(* IEC 61131-3 sources: ml2plc/examples/models/structured_text (part 7) *)

    weights_2 : ARRAY[0..3071] OF REAL := [-0.079738, -0.018148, -0.039603, 0.086091, 0.087780, 0.006551, -0.070254, -0.061014, -0.002917, -0.104361, -0.050675, -0.028002, -0.028302, -0.113236, 0.025798, -0.042125, -0.070821, -0.030886, -0.025321, 0.020352, -0.036494, -0.007489, 0.010150, 0.002465, 0.038335, -0.010082, -0.012631, -0.130657, -0.057749, -0.014712, 0.001941, 0.017731, 0.037307, 0.060894, -0.052816, -0.038803, -0.026264, 0.004428, 0.007999, -0.071385, 0.019978, -0.025107, 0.043303, -0.056437, 0.018136, -0.004926, -0.015582, -0.040352, -0.046320, -0.051167, -0.108342, 0.061847, 0.019535, 0.024186, -0.009612, 0.051589, 0.040419, 0.004677, -0.047156, 0.011391, 0.001568, -0.006703, -0.040582, -0.044892, -0.000777, -0.114299, 0.015176, 0.022018, -0.082290, -0.099898, -0.005333, -0.000085, 0.033593, -0.100384, -0.031339, -0.014356, -0.022256, -0.006458, -0.017672, -0.016220, 0.017575, -0.003964, 0.001504, -0.101623, 0.084646, -0.162545, 0.018226, 0.046139, -0.158154, -0.011727, 0.051997, 0.013728, 0.037309, 0.037653, -0.015994, -0.013833, 0.016918, 0.072840, 0.002249, 0.021758, 0.007330, -0.005101, 0.041748, 0.049668, -0.053153, -0.059272, 0.053023, -0.004963, -0.038369, -0.042376, -0.062836, 0.007027, 0.000628, 0.064942, 0.011186, 0.136276, -0.175093, 0.033480, -0.137850, -0.093329, 0.028996, 0.027738, 0.027495, 0.066908, -0.138166, -0.062207, 0.031390, 0.016039, 0.006747, 0.041813, -0.052656, -0.001730, 0.027697, -0.081471, -0.040016, 0.029091, -0.036192, 0.076833, -0.040911, 0.054524, 0.042687, 0.004638, 0.028443, -0.015942, 0.033767, -0.010835, 0.015542, -0.054845, 0.070825, -0.016626, 0.127162, -0.148593, -0.091221, 0.026570, 0.028940, 0.004587, 0.004252, 0.003949, 0.009750, 0.054379, -0.041042, 0.045454, -0.025805, 0.023543, 0.049444, 0.016239, 0.092608, 0.023911, 0.023148, 0.032898, 0.001731, 0.000178, -0.026304, -0.012553, -0.038693, 0.011086, -0.086358, -0.012758, -0.095144, -0.067500, 0.058514, 0.063057, -0.007906, 0.011515, 0.033430, 0.059557, 0.016737, -0.005871, 0.035359, -0.028117, -0.041617, -0.050268, -0.022380, -0.027072, 0.032683, 0.043795, -0.096440, 0.061286, 0.063994, -0.063137, 0.037471, -0.013500, 0.031420, 0.048276, 0.039014, -0.015300, -0.075964, 0.020676, -0.004749, -0.019730, 0.011212, -0.001377, -0.030352, -0.032305, -0.070925, -0.009115, 0.002307, 0.015789, 0.015110, -0.050587, -0.070865, -0.040802, -0.023738, -0.059662, -0.066688, 0.087581, -0.040323, 0.046836, 0.033400, 0.041713, 0.020144, 0.004004, 0.043881, 0.012120, 0.006567, -0.047181, -0.036415, 0.020897, -0.051205, -0.018987, 0.062641, -0.077042, -0.050492, -0.009248, -0.029647, -0.028774, 0.034574, 0.026711, 0.018497, -0.078291, 0.000750, 0.036981, -0.032199, -0.046941, -0.071874, 0.018149, 0.047391, 0.036563, 0.071201, -0.046533, -0.008354, -0.010784, -0.023974, 0.000798, -0.028594, -0.005823, -0.023141, 0.052901, -0.046988, 0.042628, -0.015610, 0.017471, -0.006060, -0.071074, 0.009814, 0.028930, -0.065885, 0.004670, -0.017008, 0.040985, 0.017000, 0.023364, 0.017848, -0.010962, -0.012304, 0.056049, -0.024912, 0.058021, 0.021300, -0.043819, 0.032877, -0.103125, -0.033170, 0.024651, -0.021986, -0.040304, -0.039152, -0.070680, 0.030104, -0.009235, -0.000069, 0.079351, -0.069846, -0.013240, -0.029293, 0.010581, 0.024807, -0.148111, 0.011108, -0.006310, -0.019430, -0.007536, -0.023961, -0.058471, 0.062022, 0.030894, -0.126689, 0.014609, 0.080879, 0.077431, 0.049936, 0.057099, 0.035921, -0.095284, -0.055119, 0.003187, -0.032224, -0.023817, -0.013887, -0.012151, 0.081267, 0.002542, 0.031867, -0.038254, -0.038660, -0.020785, -0.042612, 0.006728, -0.017310, 0.096375, 0.003581, -0.078691, -0.015241, -0.028676, -0.030744, -0.033101, 0.000131, -0.012343, 0.062320, 0.038591, 0.005985, 0.042647, 0.020790, -0.148493, -0.026770, -0.021416, 0.007593, 0.007429, 0.052336, 0.045379, 0.011810, -0.062384, -0.009387, -0.031314, -0.007850, -0.031340, -0.022787, -0.021615, -0.002952, 0.056798, -0.033256, -0.040985, 0.044623, -0.019729, 0.040531, -0.009346, 0.074998, -0.115437, -0.030462, 0.063818, -0.056515, -0.067471, -0.070527, -0.068923, 0.035830, -0.052215, 0.016097, -0.058752, -0.008437, -0.024348, -0.049775, -0.009136, 0.091045, -0.007442, 0.001373, 0.006184, -0.011116, -0.078380, -0.038023, 0.059468, 0.069133, -0.014606, 0.013753, -0.061774, -0.093455, 0.029663, 0.027740, -0.001149, -0.067593, -0.015326, -0.102692, -0.049083, 0.090420, 0.002557, -0.059069, -0.012321, -0.038434, 0.014221, -0.014216, 0.018523, -0.042681, -0.041700, -0.040420, -0.076709, 0.110400, -0.077629, 0.030365, -0.005439, -0.079538, 0.055336, -0.009865, -0.003723, 0.014380, 0.023391, 0.054367, -0.023334, -0.057359, -0.021853, 0.008266, 0.039793, -0.024814, 0.010200, 0.029996, 0.015745, 0.091485, -0.035740, -0.081574, 0.032012, -0.086098, -0.021267, 0.015700, 0.026081, 0.053181, -0.011251, 0.002709, -0.017904, 0.033816, 0.041051, 0.020465, 0.044652, 0.033611, 0.034061, 0.024369, 0.022682, 0.059236, -0.037332, -0.024917, 0.081315, -0.044821, -0.039097, -0.022489, -0.018730, 0.012051, 0.015785, -0.084618, -0.059913, -0.096852, -0.002574, 0.033606, 0.032488, -0.003370, 0.021578, -0.006767, -0.090289, -0.041813, -0.130182, 0.018747, 0.026137, 0.015171, -0.023929, 0.052123, 0.021562, 0.021162, 0.021938, 0.011171, 0.021531, -0.086418, -0.003059, -0.011323, -0.022397, -0.067489, 0.024647, -0.066202, -0.063597, 0.062780, -0.004904, -0.087994, 0.028886, 0.005226, 0.009394, 0.023893, -0.172482, 0.027981, -0.000874, -0.021041, 0.003634, -0.079888, 0.033055, 0.054404, -0.056195, 0.015224, -0.133033, 0.047975, 0.015738, -0.021576, -0.054744, 0.002027, -0.013741, 0.044122, 0.026994, 0.024536, -0.007580, -0.015404, -0.107729, -0.034309, -0.001584, 0.042350, 0.027646, -0.121416, -0.070898, -0.072544, -0.011634, 0.046801, 0.015250, 0.011697, -0.042356, 0.051572, -0.065324, -0.191804, -0.028124, -0.033760, -0.010601, 0.017532, 0.028585, 0.076237, 0.019598, -0.024975, 0.031572, 0.007237, 0.067220, -0.013791, 0.011680, -0.021350, -0.002438, -0.010119, 0.007116, 0.012485, 0.033664, -0.036864, 0.001408, -0.026694, 0.001947, 0.016282, -0.066502, 0.009839, -0.001735, -0.113909, -0.072450, -0.062847, -0.037870, -0.087260, -0.038781, 0.025079, 0.017764, 0.033688, 0.025043, 0.022624, 0.009969, 0.003986, 0.063781, -0.007597, -0.049656, -0.020397, 0.032632, -0.004652, -0.053405, 0.016837, -0.047092, -0.069625, -0.009141, 0.049571, -0.130610, -0.021009, -0.011360, -0.012663, 0.021738, -0.067932, 0.006787, 0.059326, -0.049219, 0.003835, 0.015163, -0.035672, 0.065436, 0.048310, 0.019535, -0.004874, -0.004026, -0.046664, 0.004075, -0.018004, 0.062538, -0.018076, 0.120624, 0.006330, -0.035533, -0.001704, 0.098006, -0.055209, 0.036600, -0.036076, -0.020109, -0.035783, 0.008194, -0.015533, 0.016326, 0.022006, -0.018952, -0.034037, -0.049213, 0.015440, -0.009457, 0.017274, 0.000384, 0.007341, -0.160581, 0.030154, 0.008035, -0.007849, 0.056014, -0.113214, 0.077642, 0.063506, 0.001735, 0.018061, 0.018220, -0.002619, -0.010912, -0.062883, -0.026722, 0.070398, -0.116190, 0.085913, -0.087937, -0.015124, 0.005143, 0.021489, 0.020521, -0.021773, -0.069295, 0.062971, 0.026118, -0.029942, -0.033439, 0.014745, 0.046682, 0.034252, -0.120951, -0.110139, 0.009602, 0.082952, 0.048315, -0.085385, -0.020953, -0.139512, 0.002793, -0.028055, 0.091898, -0.117436, 0.053042, 0.027182, -0.039500, 0.038787, 0.091544, -0.076503, 0.011879, -0.034063, -0.050604, -0.004790, 0.025791, -0.030319, -0.035485, 0.134135, -0.001677, -0.027659, -0.029312, -0.106740, -0.117414, -0.026257, 0.013410, 0.010286, -0.065646, 0.016381, 0.007505, -0.076213, -0.074846, -0.070787, -0.024315, -0.034917, -0.028188, -0.157352, 0.018341, 0.018372, 0.039563, -0.005741, -0.038507, 0.033666, -0.025694, 0.044418, -0.004166, -0.040944, -0.106082, 0.057489, -0.113991, 0.063756, 0.037792, -0.115992, -0.043843, 0.043046, 0.043409, 0.049411, 0.039022, -0.046223, -0.072060, -0.018096, 0.016482, -0.017984, -0.032877, -0.192162, 0.061553, -0.002279, -0.046261, -0.023567, -0.005539, 0.000766, -0.027724, -0.014538, 0.023718, 0.031273, -0.018895, 0.015350, -0.051778, 0.004703, 0.011070, 0.042819, -0.055612, 0.034337, 0.011549, 0.002896, 0.022180, -0.012742, -0.029711, -0.013315, 0.005108, -0.011043, 0.054103, -0.057152, -0.048314, -0.053929, 0.024708, 0.034920, 0.009985, -0.004260, -0.020098, -0.008566, 0.005943, -0.020162, -0.029077, -0.003532, -0.060852, -0.053032, -0.041148, 0.025615, 0.037711, -0.035874, -0.036773, -0.008593, 0.003211, 0.020049, 0.023300, -0.120894, 0.054418, 0.073206, 0.040949, -0.007438, -0.026906, 0.001979, 0.003925, -0.039093, -0.013398, 0.002608, 0.046654, -0.063028, 0.097928, -0.104563, -0.090482, -0.059745, 0.017705, 0.019805, -0.018141, -0.085523, -0.068505, -0.010553, -0.018658, -0.071978, 0.016467, 0.030054, 0.044513, 0.042139, 0.017734, 0.014650, 0.011766, 0.031557, -0.030363, 0.027465, -0.019329, 0.025843, -0.029637, 0.021589, 0.043354, -0.035083, -0.000107, -0.005062, -0.082215, -0.061146, -0.065887, -0.005305, 0.003747, 0.005892, 0.064349, -0.134454, -0.039398, 0.019579, 0.040492, 0.059368, -0.020607, 0.072053, 0.020348, -0.065895, -0.010689, -0.052814, -0.004183, 0.050602, 0.008220, -0.016171, -0.156647, -0.035983, -0.015830, -0.020916, 0.070798, 0.060670, 0.036338, 0.014581, -0.063205, -0.040267, -0.040092, -0.031721, -0.042686, -0.030786, 0.047541, -0.060490, 0.008227, -0.065795, 0.157321, -0.063524, -0.010021, 0.000008, -0.025935, -0.029633, -0.007435, -0.024748, 0.011676, 0.003735, -0.002965, 0.011383, 0.022123, 0.085860, -0.013978, 0.004451, -0.016815, 0.100267, -0.052584, -0.040059, 0.017191, -0.034235, -0.047621, 0.047988, 0.030696, 0.008182, 0.053458, -0.010529, 0.003663, 0.093127, -0.025486, 0.010229, 0.011255, 0.053184, 0.039015, 0.019475, -0.033527, -0.046627, 0.020910, 0.054180, -0.021971, -0.076144, -0.041172, -0.077657, -0.023235, -0.159827, 0.061509, 0.011674, -0.047834, -0.032448, -0.085723, -0.030836, -0.005105, -0.045978, 0.051450, 0.047300, -0.054793, 0.069438, -0.053058, -0.008259, 0.037206, 0.017042, 0.012406, 0.029182, -0.013802, 0.055116, -0.026872, -0.013121, 0.008830, 0.022967, -0.112740, 0.015240, 0.035079, 0.034490, 0.032152, 0.027436, -0.037881, 0.013463, 0.007487, -0.011331, 0.041363, -0.072914, -0.005484, 0.092356, 0.049594, 0.011084, 0.012504, 0.042078, -0.052556, -0.023682, -0.127495, -0.035744, 0.009192, -0.015778, -0.018911, 0.019519, 0.015076, 0.064946, 0.005913, -0.041631, 0.005621, 0.000135, 0.013980, 0.035558, -0.001797, -0.019272, -0.049151, -0.017861, -0.030677, -0.089500, -0.073268, -0.018640, -0.010916, -0.120443, 0.113037, -0.106950, 0.007440, 0.002082, 0.017529, 0.122488, -0.004168, -0.061979, 0.007902, -0.067233, 0.060663, -0.056892, -0.067239, -0.040469, -0.067240, 0.031808, -0.011052, 0.004720, -0.144488, -0.011898, -0.015811, 0.000597, 0.039404, -0.001388, 0.037090, -0.045151, 0.004902, 0.019942, 0.042480, -0.019048, 0.015990, 0.011926, 0.032038, 0.015182, 0.060560, 0.012875, 0.012309, -0.001427, 0.026395, 0.027359, 0.021883, -0.077739, -0.032637, 0.016118, 0.079860, -0.007848, 0.055546, 0.038951, -0.024144, -0.009935, 0.048732, -0.040901, -0.005186, 0.002320, 0.015519, 0.007067, 0.034431, 0.025231, -0.025804, -0.030049, 0.053530, -0.004932, -0.061164, -0.036319, 0.009787, 0.035636, 0.025358, 0.037610, 0.032730, 0.021214, -0.001584, -0.001824, 0.055127, 0.028759, 0.003438, 0.007361, 0.033248, -0.047966, -0.043201, -0.043345, 0.032240, -0.094347, -0.038789, -0.010204, 0.058107, 0.047473, 0.035086, -0.028541, 0.036375, 0.042261, -0.074968, 0.004356, 0.006226, 0.044874, 0.031667, -0.019203, 0.007147, -0.021969, 0.002657, 0.039430, -0.021067, 0.032226, 0.010131, 0.022601, 0.030890, 0.022729, 0.023010, 0.118499, -0.018482, 0.028922, -0.001738, 0.034271, -0.028747, 0.038946, 0.005030, 0.002307, 0.039449, 0.047234, -0.117320, -0.008865, 0.090959, -0.040584, -0.007000, 0.029122, -0.024144, 0.019800, 0.046470, 0.005309, -0.040488, -0.039916, -0.023335, -0.060801, 0.055213, -0.162919, -0.057773, 0.033540, -0.018969, 0.077878, 0.068904, -0.069045, -0.063349, -0.049359, -0.029544, 0.018831, -0.009165, 0.011261, 0.013990, 0.020510, 0.031716, 0.055892, -0.129224, -0.008290, 0.005706, -0.029417, -0.017326, -0.013960, -0.066511, -0.015190, -0.012143, -0.047921, 0.006963, 0.128978, -0.102790, -0.100553, 0.023065, 0.008552, -0.147233, -0.059028, -0.011403, 0.010332, -0.025088, -0.005222, -0.033179, 0.052132, -0.054748, -0.065277, -0.049472, -0.030080, -0.018076, 0.024384, 0.000906, 0.034000, 0.038237, -0.047924, 0.016248, -0.119984, -0.023678, -0.017132, -0.025957, -0.081225, -0.019621, 0.010821, -0.017947, -0.012759, 0.012802, 0.014833, -0.195305, 0.019450, -0.045534, -0.090271, 0.022506, 0.018222, 0.034140, 0.050362, -0.000892, 0.009510, 0.001972, 0.010199, 0.016216, 0.018275, 0.016543, -0.007930, -0.029494, -0.031427, -0.050046, -0.001758, 0.013238, 0.049629, 0.089262, 0.054348, -0.143622, 0.015351, 0.040831, 0.005209, 0.023357, 0.013658, 0.003482, 0.021988, -0.024363, 0.046214, -0.036009, -0.023145, -0.057607, 0.040554, 0.013757, 0.000345, -0.039764, 0.015288, 0.023860, -0.021972, 0.019933, 0.008924, -0.007245, -0.015349, -0.070772, -0.043277, -0.037041, -0.065642, 0.037743, 0.031915, 0.065512, -0.057646, 0.009085, 0.005462, -0.037111, -0.025648, -0.014509, 0.048984, -0.062467, 0.008350, 0.020535, 0.024359, -0.135527, 0.061525, 0.067536, 0.014712, -0.022363, -0.054568, -0.010573, 0.018616, 0.130626, -0.161028, 0.018211, -0.074025, -0.056558, 0.062900, 0.058391, 0.012466, 0.039785, -0.051570, -0.024763, 0.011717, -0.020121, -0.005154, 0.022717, -0.085085, -0.004483, 0.006267, 0.056714, 0.018517, -0.013750, -0.056651, 0.014559, -0.083757, 0.034585, 0.062090, 0.025170, 0.205134, 0.008425, 0.045037, -0.007797, -0.014811, 0.047300, -0.050895, 0.042679, -0.002057, -0.027680, -0.009246, 0.049523, -0.009177, 0.021952, 0.010654, 0.016540, 0.025965, 0.025313, 0.016024, -0.001483, 0.057466, -0.050435, 0.028719, 0.011265, 0.083745, -0.071478, -0.015540, -0.011341, -0.030182, 0.044617, 0.009245, -0.005794, 0.020001, 0.006360, 0.026399, 0.021226, 0.023264, -0.122019, -0.023946, -0.041825, -0.045827, -0.000447, -0.100240, 0.011886, -0.077250, -0.046740, 0.030560, 0.025529, -0.057003, 0.056144, 0.028810, 0.000188, 0.019141, 0.033223, 0.048171, -0.012389, 0.034053, 0.002163, 0.026426, -0.006897, 0.013791, 0.023153, -0.074924, -0.054218, -0.068241, 0.025634, 0.041547, 0.038397, 0.033425, -0.020355, 0.000451, -0.002249, -0.008985, -0.015632, 0.029519, 0.038687, 0.015203, -0.051157, -0.026777, -0.002135, -0.011332, -0.007479, 0.028762, 0.006724, 0.023565, 0.015143, 0.024486, 0.030722, 0.024783, 0.039658, 0.028045, 0.023870, -0.008962, -0.050171, -0.022057, 0.016545, -0.014858, 0.034915, -0.021609, 0.009053, 0.010257, -0.103685, -0.036916, 0.002683, -0.006185, -0.037673, -0.031957, -0.033120, -0.022922, 0.015500, 0.012787, -0.045898, -0.051086, 0.003612, -0.061041, -0.013488, 0.040657, 0.004496, -0.033017, 0.021011, 0.055691, 0.014075, 0.003228, -0.024891, -0.007397, -0.001558, -0.039652, 0.024171, -0.018825, 0.078651, -0.011215, 0.004297, -0.030173, -0.018809, 0.012098, -0.097526, 0.005449, 0.110859, -0.032199, -0.073718, 0.071248, -0.043038, 0.021144, 0.023286, 0.034068, 0.034989, 0.002830, -0.042828, 0.004453, -0.000080, -0.013178, -0.014562, -0.096036, -0.023655, 0.030455, -0.002976, 0.016773, 0.041034, 0.052148, -0.178205, 0.053925, 0.068062, 0.005427, 0.023584, 0.031574, 0.039421, -0.010705, -0.024920, -0.026871, 0.025332, 0.042819, -0.012192, -0.005105, 0.017539, 0.000350, 0.032542, -0.055655, 0.038161, 0.042798, 0.027429, -0.029599, 0.007941, 0.015036, 0.023611, 0.011365, -0.099722, 0.049381, 0.037109, 0.025719, 0.021033, 0.010652, 0.005350, -0.021872, 0.000794, -0.014634, 0.048023, -0.002829, -0.036040, -0.073145, -0.048980, -0.000315, -0.027606, 0.005141, 0.078039, 0.037170, 0.026744, -0.030886, -0.044456, -0.015249, -0.028043, -0.001040, 0.014369, -0.048288, -0.003488, -0.012115, 0.021661, -0.008801, -0.058470, -0.002832, -0.045678, -0.037944, 0.011971, 0.002273, 0.021211, -0.044958, -0.106527, -0.035682, -0.017779, 0.054865, 0.018123, -0.026699, 0.049155, 0.056578, 0.006985, 0.015589, 0.055782, -0.040051, -0.045889, -0.002303, -0.011842, 0.126801, -0.046605, -0.060350, -0.033177, -0.054554, -0.005002, -0.021295, -0.017539, -0.025155, -0.026726, -0.021714, 0.028631, 0.055339, 0.022541, 0.080181, 0.010012, 0.017050, -0.007285, -0.013838, 0.016927, 0.053222, 0.006573, -0.043980, -0.021879, -0.109481, -0.012588, 0.037288, 0.024495, 0.035572, 0.075180, -0.089142, 0.077327, 0.095499, 0.006064, -0.090066, 0.016709, 0.036630, -0.037648, 0.030914, 0.016806, -0.014977, 0.032918, -0.061974, -0.017286, 0.032718, 0.135538, -0.101437, 0.002422, 0.087499, 0.019634, 0.048253, 0.059520, 0.053130, 0.057759, -0.038040, -0.017170, 0.011931, -0.022979, -0.042300, -0.011427, -0.011862, -0.004407, 0.006195, 0.032012, 0.037610, 0.044604, -0.072595, 0.041505, 0.023459, -0.058261, -0.018178, 0.078624, 0.021010, -0.040663, -0.062273, -0.061405, -0.056587, -0.088124, 0.011836, -0.086923, 0.009684, 0.044435, 0.001880, 0.013791, -0.044213, -0.003511, 0.081981, -0.104622, 0.023257, -0.017744, -0.075598, 0.042589, 0.035769, 0.000795, 0.016077, -0.065667, 0.062825, 0.041799, 0.016270, 0.030678, 0.011039, -0.105255, -0.004143, 0.059784, -0.021172, 0.019785, -0.028642, -0.004309, -0.056212, -0.078287, -0.022731, -0.056815, -0.005105, -0.014022, -0.031311, -0.023550, -0.021998, -0.024260, 0.032362, 0.064688, -0.091890, -0.059349, -0.005558, -0.011701, -0.017914, -0.000725, 0.008533, 0.017962, -0.054810, -0.007925, -0.006631, 0.027688, -0.030454, 0.004947, -0.001828, 0.054848, -0.188402, -0.020981, 0.000641, 0.055269, 0.026539, -0.012360, 0.038757, -0.021594, 0.028357, 0.039710, -0.073920, -0.094747, -0.064172, -0.044126, 0.019130, 0.067423, 0.000959, -0.016326, 0.003039, 0.007727, 0.011799, 0.006578, -0.004746, 0.042672, -0.003960, 0.044675, 0.036238, 0.035630, 0.032696, 0.031020, -0.004627, 0.013475, 0.042956, -0.052501, -0.016311, -0.051736, 0.003689, 0.056814, 0.032506, 0.051707, 0.133479, -0.042669, 0.022440, 0.022948, -0.023296, -0.005525, 0.051002, 0.052883, 0.058544, -0.050477, 0.044311, 0.002172, 0.083715, -0.039275, 0.057967, 0.068556, 0.037423, -0.060565, 0.038015, -0.078545, 0.043739, -0.003802, -0.017818, -0.010219, 0.150024, -0.010153, -0.101539, -0.001109, -0.014247, -0.016844, 0.033372, 0.014056, 0.016519, 0.007482, -0.027599, -0.007664, 0.013053, -0.004768, -0.008083, 0.007597, -0.040281, -0.024178, 0.005960, 0.037884, 0.033172, -0.030735, -0.042964, -0.030635, -0.024636, 0.008905, -0.002768, 0.053170, -0.072516, -0.081345, 0.018499, 0.027379, 0.003028, -0.006458, -0.105476, -0.060001, -0.019271, -0.031725, 0.087183, -0.088419, -0.028217, -0.002698, -0.003315, -0.055869, 0.031687, -0.044833, -0.055949, -0.074364, -0.020587, -0.140201, 0.001538, 0.014761, -0.017415, -0.050676, -0.050461, 0.083559, -0.054638, -0.027387, -0.076291, -0.037181, -0.010422, -0.042042, -0.012635, 0.032873, 0.037906, 0.047499, 0.019249, -0.099218, -0.008168, 0.054566, -0.090759, 0.029319, -0.009164, -0.025257, -0.004178, -0.019100, -0.057294, -0.057693, -0.022269, -0.008831, 0.000688, 0.077182, -0.007420, 0.001672, -0.002048, -0.071018, 0.040179, -0.111050, -0.049216, 0.003540, -0.040745, -0.038487, -0.064390, -0.110880, 0.050489, 0.030086, 0.041917, 0.078558, -0.107200, -0.026824, 0.015360, 0.016766, 0.013769, 0.007341, 0.063267, 0.042176, 0.043688, 0.041885, -0.127719, 0.003388, 0.026274, -0.007837, -0.097381, -0.004769, 0.055554, 0.009136, -0.052764, -0.039822, 0.087266, -0.192491, 0.049151, 0.030375, 0.035820, -0.009659, -0.057846, -0.065094, -0.046896, -0.057456, -0.017067, -0.034092, -0.007246, 0.008380, 0.027120, 0.070289, -0.055207, 0.043841, 0.029015, 0.010738, -0.056403, -0.058787, -0.057282, 0.019799, 0.101903, -0.144661, 0.014157, -0.101370, 0.035069, 0.009934, -0.005132, -0.034092, 0.014860, -0.012129, 0.041441, 0.042958, 0.026968, 0.011155, -0.007552, -0.012508, -0.002572, 0.016272, -0.011616, 0.010629, -0.009160, -0.015472, 0.015415, 0.029885, -0.010060, 0.002749, -0.072919, -0.066665, -0.041343, 0.039695, -0.053709, -0.021016, -0.000614, 0.067261, 0.036065, -0.032962, -0.037148, -0.057983, 0.006014, 0.072962, 0.066036, 0.074045, 0.026112, 0.000779, 0.083515, -0.066614, 0.008478, -0.002375, -0.044657, -0.031095, -0.013031, 0.010733, -0.018030, 0.023650, -0.037599, 0.037502, 0.014425, 0.009555, 0.009053, -0.002985, 0.028003, 0.051038, 0.018547, 0.068332, -0.010430, 0.007832, 0.004124, 0.015459, 0.053690, 0.029809, 0.060038, -0.040707, 0.039347, -0.010417, -0.012356, -0.001695, 0.023034, -0.046593, -0.118021, 0.065954, 0.044816, -0.050910, 0.026081, 0.010554, 0.001999, -0.009056, 0.028741, 0.024808, 0.007134, 0.037890, 0.039553, 0.028437, -0.013596, -0.036495, -0.022982, 0.027081, -0.058788, -0.010266, -0.229805, -0.063225, -0.004700, 0.079670, -0.097898, 0.025573, 0.023837, -0.029241, -0.006460, 0.077259, 0.051649, 0.028394, -0.004598, 0.030752, -0.003841, 0.006880, -0.057608, -0.027399, -0.062937, -0.021952, -0.030290, 0.039727, 0.044383, 0.085802, -0.007403, -0.026491, -0.028395, -0.056531, -0.036996, -0.070584, 0.069473, -0.116761, -0.036883, -0.033294, -0.024618, -0.026149, -0.002657, -0.055080, -0.082606, 0.007050, 0.012350, -0.047867, -0.050522, 0.139970, 0.050096, 0.054879, 0.004056, 0.014902, 0.011027, 0.002136, 0.070084, 0.012674, -0.050863, -0.003282, 0.000134, 0.028618, 0.033623, 0.000763, -0.034382, -0.026524, -0.036297, -0.031225, -0.033303, 0.008783, 0.014384, 0.038812, 0.045117, 0.014172, -0.054809, -0.005565, -0.099740, -0.051121, -0.032616, -0.030484, -0.012884, -0.021194, -0.076313, -0.063640, -0.042839, -0.008553, -0.065287, 0.017557, -0.005521, -0.004356, 0.035749, -0.040603, -0.022183, -0.032807, -0.054063, -0.013052, 0.052090, -0.016355, 0.025171, -0.008166, 0.016264, 0.027828, -0.020940, -0.031619, -0.028913, 0.009505, -0.008992, -0.004273, 0.005117, 0.062502, 0.034384, -0.021784, -0.011864, -0.073795, 0.010463, -0.050705, 0.005860, 0.055013, -0.059139, 0.003764, 0.027440, 0.016377, 0.009504, 0.015080, 0.015725, 0.067479, 0.089536, 0.022483, -0.030345, 0.025729, 0.024267, 0.023434, 0.011054, -0.056527, 0.045667, -0.011390, -0.036648, -0.017359, -0.073089, -0.064995, -0.026360, -0.112975, 0.014516, -0.053314, -0.043682, -0.025288, 0.032010, 0.021024, -0.088265, 0.026747, 0.036819, -0.161553, -0.170717, 0.007788, 0.031794, 0.032223, 0.038833, 0.004319, -0.101911, 0.020677, 0.025928, 0.008587, 0.040665, 0.021545, -0.017421, -0.015369, -0.014964, -0.025905, 0.004569, 0.048798, 0.048843, -0.067144, 0.008329, 0.007224, 0.057075, 0.096059, -0.165318, -0.059617, 0.060519, 0.047643, -0.061039, 0.045086, 0.061249, 0.216103, -0.100665, -0.149878, -0.004593, -0.076908, -0.009678, 0.027603, 0.008345, -0.030318, -0.088064, -0.009970, 0.014668, 0.008051, 0.040958, -0.057137, -0.015193, -0.038329, -0.014315, 0.040159, 0.005071, -0.056252, -0.025981, -0.018578, 0.011800, 0.036899, -0.039913, -0.002179, 0.013237, 0.016750, 0.015171, -0.018277, 0.013945, -0.007538, -0.023018, -0.026236, -0.004053, 0.028176, 0.031779, 0.040546, -0.080991, 0.071929, 0.038683, 0.009296, 0.003681, -0.036370, 0.017538, 0.014322, 0.000090, 0.044998, 0.057049, 0.013201, 0.004392, -0.007755, -0.012693, -0.022717, -0.004545, -0.049206, 0.019760, 0.044115, -0.000525, 0.045303, 0.000497, 0.035163, 0.005653, 0.045240, 0.003727, -0.070555, 0.032291, 0.008739, 0.019656, 0.009403, -0.019270, 0.054355, -0.130183, 0.029607, -0.029557, 0.029361, 0.048000, -0.131765, -0.026280, -0.112344, -0.016534, -0.017396, 0.055342, 0.007255, 0.002500, 0.019163, 0.006458, 0.005560, 0.032867, -0.155293, 0.083058, -0.058361, 0.001098, 0.025701, -0.022830, -0.021569, -0.027672, -0.010628, 0.016473, 0.033767, 0.025464, 0.124101, -0.000884, -0.072848, -0.053164, 0.046359, 0.026941, -0.035541, -0.044423, -0.034902, -0.082594, -0.056229, -0.039919, -0.064250, -0.003669, -0.020732, -0.033810, -0.005944, 0.052929, 0.022141, 0.024940, -0.062812, -0.043056, -0.025592, -0.011451, 0.046149, -0.070122, 0.046039, 0.057248, -0.147282, -0.016161, -0.064449, -0.062920, -0.011957, -0.047200, -0.032719, -0.068744, -0.018227, -0.013996, 0.019577, 0.070230, -0.001122, 0.003156, -0.004815, -0.019025, -0.059807, -0.043167, -0.097361, -0.031011, -0.013155, -0.003375, -0.068266, 0.000515, -0.043310, -0.028366, -0.019327, -0.028505, -0.018100, -0.042574, -0.048828, -0.032464, 0.035071, 0.001615, -0.016472, 0.122361, -0.175405, 0.016869, -0.049321, -0.049486, -0.053595, 0.038521, -0.007626, -0.071877, 0.047651, -0.007771, 0.051924, -0.029978, -0.047229, -0.033511, 0.015380, 0.052650, -0.071036, -0.028013, 0.014148, -0.022484, -0.031536, -0.034461, -0.039607, -0.165174, -0.039282, 0.012603, 0.008545, 0.048225, 0.015458, 0.010238, 0.016575, -0.014633, -0.061731, -0.028572, -0.015910, -0.050669, -0.010256, -0.051820, -0.030456, 0.001819, 0.009222, 0.001152, -0.068290, -0.015510, 0.002223, -0.020006, -0.027246, 0.004222, 0.054849, 0.049251, 0.032987, -0.111734, -0.100253, 0.014001, -0.104118, 0.051836, 0.015181, -0.032367, -0.025997, -0.091562, -0.046772, 0.018370, 0.156002, -0.137137, -0.033829, -0.099663, -0.002590, 0.007428, -0.015988, 0.047072, 0.001561, 0.010310, -0.005918, -0.021363, 0.019911, -0.040275, 0.037233, 0.033426, -0.037623, 0.002218, -0.014229, -0.011679, -0.003373, 0.007235, 0.022227, -0.027489, 0.008246, -0.018292, 0.030887, -0.016768, -0.013755, -0.015357, -0.031411, 0.029860, 0.008441, 0.012850, 0.000829, 0.050036, 0.016729, -0.057398, -0.058280, -0.032134, 0.008055, 0.003189, -0.045665, -0.062002, -0.060869, 0.017901, 0.043825, 0.074501, -0.101529, 0.038794, -0.027028, -0.006740, 0.015007, -0.005359, 0.051557, 0.009424, 0.059670, -0.066454, 0.012280, -0.012073, -0.030648, -0.074662, 0.047514, 0.014376, 0.040649, 0.011516, -0.048052, -0.046850, 0.072419, 0.002600, 0.070362, -0.013911, -0.059027, -0.062221, 0.017670, 0.082880, -0.053215, -0.035223, -0.004333, 0.015831, 0.004593, 0.016349, 0.031053, -0.034744, 0.001690, 0.074972, 0.014751, 0.003123, 0.058507, 0.019019, 0.024827, 0.106503, -0.053284, -0.020871, -0.068255, -0.056442, -0.006431, 0.073455, -0.087469, 0.044454, -0.001962, -0.043267, 0.031325, -0.027985, 0.047023, 0.015176, -0.006171, -0.015462, -0.062765, -0.035117, -0.007201, -0.068043, -0.065041, -0.055927, -0.079111, 0.070689, 0.007429, 0.014942, -0.008060, 0.009621, 0.003918, -0.006859, 0.055769, -0.031637, 0.000228, -0.051440, -0.018303, -0.071879, -0.037196, 0.016479, -0.037846, -0.054266, 0.042683, 0.025163, 0.013933, -0.042980, -0.059458, -0.063729, 0.088301, 0.033623, -0.088517, -0.044624, -0.040706, -0.042223, 0.048527, 0.002611, -0.050081, 0.071289, 0.040366, 0.035756, -0.029064, 0.069452, 0.050530, -0.070521, -0.056548, 0.004240, 0.007107, -0.021827, 0.036275, 0.041781, -0.014992, 0.030029, 0.083748, 0.114207, -0.061393, -0.044776, -0.008920, -0.022174, 0.009187, 0.033627, 0.030427, -0.053553, -0.048855, -0.038547, -0.031399, -0.035287, -0.023365, -0.010921, 0.009142, -0.041277, 0.056985, -0.021846, 0.060162, -0.004609, 0.012687, -0.037194, 0.010759, -0.007457, -0.001846, -0.010043, -0.009611, 0.003672, -0.064335, -0.006818, 0.016462, -0.045820, 0.004625, 0.088568, 0.069543, 0.049584, 0.040205, 0.045356, 0.069874, 0.023491, -0.016608, -0.012406, -0.049791, -0.055085, 0.045394, -0.037096, -0.026840, 0.100678, 0.020555, -0.010173, -0.039356, 0.016359, -0.005669, -0.002994, -0.002770, 0.028880, -0.093406, -0.011944, -0.008557, -0.048961, -0.014940, -0.014389, -0.007846, 0.023851, -0.018251, -0.035302, 0.001411, 0.039391, 0.025447, 0.062880, 0.139204, -0.063451, 0.052854, -0.032663, -0.011902, -0.011408, 0.002335, 0.021545, 0.044586, -0.053677, 0.040654, -0.026303, 0.033930, -0.086145, -0.002936, -0.037917, 0.100404, -0.133088, 0.083269, -0.042569, 0.072479, -0.017151, -0.039370, -0.012219, -0.004206, -0.056602, -0.083909, 0.003521, -0.014192, -0.032977, 0.008703, 0.022527, 0.035428, -0.063572, -0.001681, -0.018865, -0.001556, 0.077047, 0.038923, 0.019397, -0.055465, -0.010339, 0.023785, -0.046236, -0.002640, 0.044719, 0.044637, 0.063677, -0.009018, 0.042315, -0.090560, -0.049278, -0.071467, -0.063102, -0.025515, 0.021175, 0.036242, -0.035767, 0.026336, -0.069859, 0.024859, 0.028028, 0.027595, -0.016651, -0.007722, -0.033696, 0.000070, -0.007223, -0.033072, 0.050118, -0.033982, 0.044890, 0.010682, 0.018131, 0.007655, -0.094003, 0.055888, -0.118141, 0.026367, -0.066037, -0.024128, 0.012338, -0.059165, 0.007676, 0.005133, -0.064627, -0.084559, -0.024493, 0.022035, -0.011872, -0.039371, -0.078983, 0.008282, 0.007041, 0.033947, 0.112090, 0.017122, -0.092168, 0.000329, -0.064474, -0.008359, -0.078479, -0.030748, -0.007414, -0.007756, -0.016775, -0.095148, -0.010669, 0.059292, 0.023279, -0.095457, -0.077958, -0.024279, 0.032884, 0.029683, 0.028798, 0.003811, -0.070640, -0.023708, 0.010974, 0.035563, 0.128666, -0.194970, -0.004273, 0.011050, -0.001804, 0.017223, -0.087389, 0.017226, -0.000764, -0.009369, 0.019048, 0.064953, 0.057376, 0.033859, 0.015679, 0.029313, 0.023839, -0.059955, 0.054118, 0.063973, -0.014520, 0.058390, -0.031282, -0.000189, 0.000515, 0.004418, -0.107691, -0.024868, -0.057891, 0.024555, -0.029299, 0.036922, 0.112752, 0.016979, 0.070291, -0.012889, -0.005460, 0.011498, 0.029838, 0.038815, 0.020644, -0.030950, -0.008370, -0.012246, 0.023434, -0.051213, -0.015141, -0.045205, -0.090602, -0.057723, -0.020648, 0.031079, -0.023994, -0.001400, -0.053488, -0.055061, -0.045196, 0.041105, 0.017850, -0.069851, -0.009776, -0.021581, 0.023885, -0.023427, 0.017106, -0.100083, -0.011155, -0.031993, -0.145589, -0.008524, -0.040239, 0.023660, 0.060080, 0.013866, -0.020106, 0.021282, -0.018435, 0.030530, -0.020865, 0.083572, 0.040695, 0.026287, 0.077900, 0.001829, -0.029643, 0.005312, -0.003519, -0.057242, 0.002076, -0.009702, -0.038513, -0.020878, 0.024728, -0.053036, -0.024956, 0.013848, -0.006973, -0.001531, -0.108869, 0.113928, -0.060123, 0.057967, 0.027651, 0.028142, -0.028350, -0.040685, -0.007469, 0.010442, -0.057321, 0.013665, 0.010827, -0.025913, -0.004077, 0.024542, 0.012953, -0.040154, -0.032880, -0.014401, -0.046751, 0.017235, 0.006994, 0.007214, 0.065257, -0.009963, 0.023260, 0.026583, -0.006580, 0.074270, -0.054298, -0.013688, 0.005546, 0.003241, -0.039276, 0.000855, 0.027435, 0.064403, 0.090223, -0.039380, 0.026120, -0.011682, -0.068958, 0.016665, -0.026120, -0.030531, -0.083979, -0.042100, -0.160802, -0.071336, 0.002649, -0.049153, 0.009379, 0.018974, 0.029916, -0.189163, 0.111529, 0.018877, 0.003704, 0.037302, -0.036443, 0.010205, 0.017517, 0.064199, 0.009839, 0.009605, 0.030128, 0.034517, 0.002029, -0.000867, -0.181125, 0.005753, -0.021533, -0.129864, -0.001275, -0.027567, -0.005573, 0.033724, -0.026302, -0.048262, -0.059149, -0.019389, -0.009621, -0.052161, -0.012001, -0.014082, -0.014802, 0.002952, -0.018956, -0.006534, 0.020044, -0.087776, -0.040843, -0.040039, -0.033959, -0.010779, 0.013630, 0.054790, 0.033969, -0.032992, -0.066282, -0.029683, -0.040541, 0.036804, -0.044183, -0.011512, -0.013626, 0.006024, -0.003635, 0.011609, -0.011648, -0.045873, -0.033584, -0.041106, 0.027988, -0.052191, -0.017248, 0.012694, 0.008044, -0.007954, 0.025363, -0.086099, -0.025632, 0.021677, -0.093187, -0.026642, 0.000034, -0.001859, -0.011353, -0.068031, -0.029673, -0.039027, -0.002835, -0.013504, -0.022699, 0.053803, 0.038057, 0.061807, -0.035126, 0.013087, 0.007936, 0.043549, 0.016608, 0.089125, -0.093529, -0.022182, -0.029988, 0.052475, 0.016939, 0.057350, 0.065654, -0.067515, 0.030868, 0.060191, 0.025650, 0.058997, -0.038286, -0.060195, -0.012983, 0.044122, 0.055023, 0.051873, 0.085608, -0.187042, 0.088019, -0.017523, -0.177571, 0.002488, -0.183339, -0.037920, 0.006585, 0.014863, 0.006200, -0.066613, -0.010054, -0.009553, 0.012879, 0.006688, 0.019419, 0.021633, 0.059471, -0.048183, -0.107076, 0.050837, 0.002559, 0.040617, 0.020748, -0.053189, 0.032267, 0.013923, 0.019593, 0.040685, 0.000141, 0.028513, 0.018103, -0.087549, 0.043683, -0.031831, 0.038227, 0.092663, 0.070637, 0.026814, -0.091406, -0.067131, 0.037108, -0.020395, -0.018967, 0.029855, -0.125865, -0.093615, 0.024357, 0.028657, 0.026613, -0.010095, -0.008811, -0.011117, -0.005576, -0.031336, -0.049807, 0.009479, 0.044275, 0.017381, -0.059902, -0.022112, -0.078543, -0.037100, -0.008728, -0.000979, 0.035509, -0.028954, 0.037039, 0.050164, -0.017211, 0.018334, -0.005631, -0.058840, -0.021846, -0.016327, -0.020067, -0.046736];
    bias_2 : ARRAY[0..2] OF REAL := [-0.239521, 0.362263, -0.140268];

END_VAR

VAR
    (* Buffer allocation variables *)
    buffer_0 : ARRAY[0..1023] OF REAL;
    buffer_1 : ARRAY[0..511] OF REAL;

    (* Temporary computation variables *)
    i : DINT;
    j : DINT;
    sum : REAL;
    max_val : REAL;
    exp_sum : REAL;

END_VAR

(* Layer 0: Fused Linear + RELU *)
FOR j := 0 TO 511 DO
    sum := 0.0;
    FOR i := 0 TO 4 DO
        sum := sum + input_data[i] * weights_0[i * 512 + j];
    END_FOR;
    buffer_1[j] := MAX(sum + bias_0[j], 0.0);
END_FOR;

(* Layer 1: Fused Linear + RELU *)
FOR j := 0 TO 1023 DO
    sum := 0.0;
    FOR i := 0 TO 511 DO
        sum := sum + buffer_1[i] * weights_1[i * 1024 + j];
    END_FOR;
    buffer_0[j] := MAX(sum + bias_1[j], 0.0);
END_FOR;

(* Layer 2: Fused Linear + SOFTMAX *)
FOR j := 0 TO 2 DO
    sum := 0.0;
    FOR i := 0 TO 1023 DO
        sum := sum + buffer_0[i] * weights_2[i * 3 + j];
    END_FOR;
    output_data[j] := sum + bias_2[j];
END_FOR;

max_val := output_data[0];
FOR i := 1 TO 2 DO
    IF output_data[i] > max_val THEN
        max_val := output_data[i];
    END_IF;
END_FOR;

exp_sum := 0.0;
FOR i := 0 TO 2 DO
    output_data[i] := EXP(output_data[i] - max_val);
    exp_sum := exp_sum + output_data[i];
END_FOR;

FOR i := 0 TO 2 DO
    output_data[i] := output_data[i] / exp_sum;
END_FOR;

END_FUNCTION_BLOCK
